PROGRAM MAIN
VAR
bCalibrate:	BOOL;
fFB: REAL;
fStepValue: REAL :=0.5;
fDev: REAL := 0.1;	
fCmd: REAL;
fCommandZeroError:	REAL;
fCommandSpanError:	REAL;
fFeedbackZeroError:	REAL;
fFeedbackSpanError: REAL;  
bCalibrationFinished: BOOL;
bError : BOOL;
bBusy : BOOL;
bDoubleCheck : BOOL;
fbAutoCalibration : FB_AutoCalibration;
END_VAR

fbAutoCalibration(bCalibrate:=bCalibrate,
				fFB := fFB,
				fStepValue:=fStepValue,
				fDev:=fDev,
				fBand:=0.2);

fCmd:= fbAutoCalibration.fCmd;
				
fCommandZeroError:= fbAutoCalibration.fCmdZeroErr;

fCommandSpanError:= fbAutoCalibration.fCmdSpanErr;

fFeedbackZeroError:= fbAutoCalibration.fFBZeroErr;

fFeedbackSpanError:= fbAutoCalibration.fFBSpanErr;

bCalibrationFinished:=fbAutoCalibration.bCalibrationFinished;

bError := fbAutoCalibration.bError;

bBusy := fbAutoCalibration.bBusy;

bDoubleCheck := fbAutoCalibration.bDoubleCheck;

END_PROGRAM

(* stored: Version 1.1.0.1, ProductVersion 3.1.4024.9
   POU MAIN: Id {27aaebf8-6fda-45d8-9038-d5e2a0732680}, SpecialFunc None *)
